FUNCTION_BLOCK FB_Sub1 IMPLEMENTS I_Sub1
VAR_INPUT
END_VAR
VAR_OUTPUT
END_VAR
VAR
END_VAR

{warning 'Agregar implementación de método'}
METHOD metodo_base1 : BOOL
END_METHOD

{warning 'Agregar implementación de método'}
METHOD metodo_base2 : BOOL
END_METHOD

{warning 'Agregar implementación de método'}
METHOD metodo_sub1 : BOOL
END_METHOD

{warning 'Agregar implementación de propiedad'}
PROPERTY Prop_base1 : BOOL
GET
END_GET
SET
END_SET
END_PROPERTY

{warning 'Agregar implementación de propiedad'}
PROPERTY Prop_base2 : BOOL
GET
END_GET
SET
END_SET
END_PROPERTY

{warning 'Agregar implementación de propiedad'}
PROPERTY Prop_sub1 : BOOL
GET
END_GET
SET
END_SET
END_PROPERTY

END_FUNCTION_BLOCK

(* stored: Version 1.1.0.1, ProductVersion 3.1.4024.12
   POU FB_Sub1: Id {42168c9e-7df7-4a2f-ace5-f429a736f068}, SpecialFunc None
   Method metodo_base1: Id {b113a7e6-76fd-4a40-b478-56cb170ef036}
   Method metodo_base2: Id {e45040e5-6ade-48a2-b580-855b0bea4ea4}
   Method metodo_sub1: Id {5dba1e94-8479-447b-8005-8409e037903e}
   Property Prop_base1: Id {496ff109-b6c2-4b69-a8f9-7fc556fdf205}
   Get Get: Id {52202749-733c-41c1-ae31-d33e2e9a4ce5}
   Set Set: Id {5fc175b0-9d87-4562-aac2-f6c65d206496}
   Property Prop_base2: Id {8a0e57a7-53a4-4895-81e5-62b67b00d3d3}
   Get Get: Id {175db947-67fd-4795-aa65-1f4856b128eb}
   Set Set: Id {8acc477c-6ea4-4530-bea1-959f79c2d07e}
   Property Prop_sub1: Id {adde8640-1e64-4d54-b784-42e65ed94ce2}
   Get Get: Id {2043f8fc-8550-4456-95e8-72672f1969de}
   Set Set: Id {49dc2498-1626-4a47-a8c5-8b2dfa424ae2} *)
